NAMESPACE PackedLine
ORGANIZATION_BLOCK Main_PackedLine
TITLE = "Main Program Sweep (Cycle)"
{ S7_Optimized_Access := 'TRUE' ; Published := 'FALSE' }
VERSION : 0.1

BEGIN
	IDB_PackedLine();

END_ORGANIZATION_BLOCK
END_NAMESPACE

